{attribute 'qualified_only'}
{attribute 'strict'}
TYPE E_HistoryDiagDevices :
(
	EL19xx		:= 0,
	EL29xx 		:= 1
);
END_TYPE

(* stored: Version 1.1.0.1, ProductVersion 3.1.4024.12
   DUT E_HistoryDiagDevices: Id {2c43444c-1a95-49d3-9354-3685ed0a72a3} *)
